// Mitsubishi GX Works2 project: 자기유지회로   PLC: Q03UDV

PROGRAM MAIN
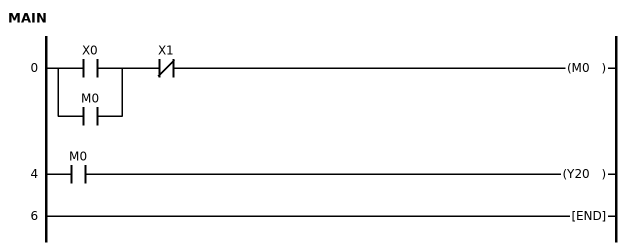
0     LD      X0
      OR      M0
      ANI     X1
      OUT     M0
4     LD      M0
      OUT     Y20
6     END
END_PROGRAM
